{attribute 'GeneratedUsingTerminal: AMI8000-0000-0016'}
{attribute addProperty BoxType "AMI8000-0000-0016"}
{attribute addProperty Id "StatuswordAT %I*UINT2"}
{attribute addProperty CRC "2604072444"}
{attribute addProperty Size "2"}
TYPE DRV_Statusword_9B36FDFC :
STRUCT
	{attribute addProperty Name "Statusword"}
	Statusword AT %I* : UINT;
END_STRUCT
END_TYPE

(* stored: Version 1.2.0.0, ProductVersion 3.1.4024.9
   DUT DRV_Statusword_9B36FDFC: Id {6d932e1f-fe8f-4f60-8323-01a49512bc73} *)
